	childCriticalErrorReaction : CHILD_CRITICAL_ERROR_REACTION;
	
	i : INT;
		
	child : IChildAutomationComponent;	

	inputDevice : IInputLeafAutomationComponent;
END_VAR
__TRY
	OnBeforeChildrenProcessInput();
__CATCH(exceptionCode)		
	exception := TOF_Core.ExceptionManager.GetLastException(
		exceptionCode := exceptionCode,
		catchPointNamespaceName := NamespaceName,
		catchPointPOUName := __POUNAME(),
		catchPointPosition := __POSITION()
	);
					
	exceptionReaction := OnHandleException(exception := exception, failedMethodName := 'OnBeforeChildrenProcessInput');

	ProcessException(
		exception := exception,
		exceptionReaction := exceptionReaction,
		exceptionSourceHint := "OnBeforeChildrenProcessInput error"
	);
__ENDTRY

FOR i := 0 TO _ChildCount - 1 DO
	child := TryGetChildByIndex(index := i);

	IF child = 0 OR_ELSE NOT child.Enabled OR_ELSE NOT __QUERYINTERFACE(child, inputDevice) THEN
		CONTINUE;
	END_IF
	
	inputDevice.ProcessInput();

	IF inputDevice.HasError AND_THEN inputDevice.Error.Severity = TOF_Core.ERROR_SEVERITY.CRITICAL THEN
		childCriticalErrorReaction := HandleChildCriticalError(childWithError := inputDevice);
		
		ProcessChildError(
			childError := inputDevice.Error,
			childErrorReaction := childCriticalErrorReaction,
			childErrorSourceHint := TOF_Core.WideStrings.Concat255(
				"Child[",
				TO_WSTRING(i),
				"](",
				inputDevice.Name,
				").ProcessInput error"
			)
		);
	END_IF		
END_FOR

__TRY
	OnAfterChildrenProcessInput();
__CATCH(exceptionCode)		
	exception := TOF_Core.ExceptionManager.GetLastException(
		exceptionCode := exceptionCode,
		catchPointNamespaceName := NamespaceName,
		catchPointPOUName := __POUNAME(),
		catchPointPosition := __POSITION()
	);
					
	exceptionReaction := OnHandleException(exception := exception, failedMethodName := 'OnAfterChildrenProcessInput');

	ProcessException(
		exception := exception,
		exceptionReaction := exceptionReaction,
		exceptionSourceHint := "OnAfterChildrenProcessInput error"
	);
__ENDTRY
END_METHOD

(*!
<summary>Processes enabled output children in slot order.</summary>
<description>
A state transition during output processing skips remaining outputs and the after-output hook.
Completed writes remain effective. A pass started in STOPPED proceeds while the branch stays in that state.
</description>
*)
METHOD FINAL ProcessOutput
VAR
	entryRevision : UDINT;
	exceptionCode : __SYSTEM.ExceptionCode;
	exception : TOF_Core.IException;	
	exceptionReaction : TOF_Core.EXCEPTION_REACTION;
	
	childCriticalErrorReaction : CHILD_CRITICAL_ERROR_REACTION;
	
	i : INT;
		
	child : IChildAutomationComponent;	

	outputDevice : IOutputLeafAutomationComponent;
END_VAR
entryRevision := _OperationalStateRevision;

__TRY
	OnBeforeChildrenProcessOutput();
__CATCH(exceptionCode)		
	exception := TOF_Core.ExceptionManager.GetLastException(
		exceptionCode := exceptionCode,
		catchPointNamespaceName := NamespaceName,
		catchPointPOUName := __POUNAME(),
		catchPointPosition := __POSITION()
	);
					
	exceptionReaction := OnHandleException(exception := exception, failedMethodName := 'OnBeforeChildrenProcessOutput');

	ProcessException(
		exception := exception,
		exceptionReaction := exceptionReaction,
		exceptionSourceHint := "OnBeforeChildrenProcessOutput error"
	);
__ENDTRY

FOR i := 0 TO _ChildCount - 1 DO
	IF _OperationalStateRevision <> entryRevision THEN
		RETURN;
	END_IF

	child := TryGetChildByIndex(index := i);

	IF child = 0 OR_ELSE NOT child.Enabled OR_ELSE NOT __QUERYINTERFACE(child, outputDevice) THEN
		CONTINUE;
	END_IF
	
	IF _OperationalStateRevision <> entryRevision THEN
		RETURN;
	END_IF

	outputDevice.ProcessOutput();
	
	IF outputDevice.HasError AND_THEN outputDevice.Error.Severity = TOF_Core.ERROR_SEVERITY.CRITICAL THEN
		childCriticalErrorReaction := HandleChildCriticalError(childWithError := outputDevice);
		
		ProcessChildError(
			childError := outputDevice.Error,
			childErrorReaction := childCriticalErrorReaction,
			childErrorSourceHint := TOF_Core.WideStrings.Concat255(
				"Child[",
				TO_WSTRING(i),
				"](",
				outputDevice.Name,
				").ProcessOutput error"
			)
		);
	END_IF
END_FOR

IF _OperationalStateRevision <> entryRevision THEN
	RETURN;
END_IF

__TRY
	OnAfterChildrenProcessOutput();
__CATCH(exceptionCode)		
	exception := TOF_Core.ExceptionManager.GetLastException(
		exceptionCode := exceptionCode,
		catchPointNamespaceName := NamespaceName,
		catchPointPOUName := __POUNAME(),
		catchPointPosition := __POSITION()
	);
					
	exceptionReaction := OnHandleException(exception := exception, failedMethodName := 'OnAfterChildrenProcessOutput');

	ProcessException(
		exception := exception,
		exceptionReaction := exceptionReaction,
		exceptionSourceHint := "OnAfterChildrenProcessOutput error"
	);
__ENDTRY
END_METHOD

(*!
<summary>Returns a borrowed child by its zero-based index.</summary>
<description>
Returns null when the entry is unavailable, the index is out of range or a nested call raises an exception.
Fatal allocation observations before or after the storage getter return null and preserve the latch for
the outer task boundary. Does not transfer ownership or extend lifetime. Getter exceptions are contained.
</description>
*)
METHOD FINAL TryGetChildByIndex : IChildAutomationComponent
VAR_INPUT
	index : TOF_Core.INT_INDEX;
END_VAR
VAR
	childStorage : REFERENCE TO ARRAY [0.._ChildCount - 1] OF IChildAutomationComponent;
END_VAR
__TRY
	IF TOF_Core.DynamicMemoryManager.HasAllocationFailed OR_ELSE index < 0 OR_ELSE index >= _ChildCount THEN
		RETURN;
	END_IF

	childStorage REF= Children;

	IF NOT TOF_Core.DynamicMemoryManager.HasAllocationFailed AND_THEN __ISVALIDREF(childStorage) THEN
		TryGetChildByIndex := childStorage[index];
	END_IF
__CATCH
	TryGetChildByIndex := 0;
__ENDTRY

IF TOF_Core.DynamicMemoryManager.HasAllocationFailed THEN
	TryGetChildByIndex := 0;
END_IF
END_METHOD

METHOD PROTECTED FINAL Validate
VAR
END_VAR
IF _Parent = 0 THEN
	TOF_Core.Exceptions.ThrowDataMemberNotSpecified(
		sourceNamespaceName := NamespaceName,
		sourceClassName := ClassName,
		sourcePOUName := __POUNAME(),
		sourcePosition := __POSITION(),
		dataMemberName := 'Parent'
	);						
END_IF

IF ChildCount > 0 AND_THEN NOT __ISVALIDREF(Children) THEN
	TOF_Core.Exceptions.ThrowDataMemberNotSpecified(
		sourceNamespaceName := NamespaceName,
		sourceClassName := ClassName,
		sourcePOUName := __POUNAME(),
		sourcePosition := __POSITION(),
		dataMemberName := 'Children'
	);
END_IF
END_METHOD

END_FUNCTION_BLOCK

// ---- AutomationComponent/Branches/ChildCriticalErrorHandlingPolicies/ChildCriticalErrorHandlingPolicies.TcPOU
(*
SPDX-FileCopyrightText: Â© 2026 Oleksandr Tiutyk <trofimich@gmail.com>
SPDX-License-Identifier: MIT
License: https://opensource.org/license/mit
*)

(*!
<summary>Provides shared singleton instances of child critical error handling policies.</summary>
*)

{attribute 'no_explicit_call' := 'do not call this function block directly'}
PROGRAM ChildCriticalErrorHandlingPolicies
VAR
	{attribute 'hide'} 
	_ClassName : STRING := __POUNAME();
	
	{attribute 'hide'} 
	_SetErrorAndStop : SetErrorAndStopAfterCriticalChildErrorHandlingPolicy; 
	{attribute 'hide'} 
	_SetErrorAndContinue : SetErrorAndContinueAfterChildCriticalErrorHandlingPolicy; 
	{attribute 'hide'} 
	_Ignore : IgnoreChildCriticalErrorHandlingPolicy; 
END_VAR

(*!
<summary>Gets the class name of the program.</summary>
*)
{attribute 'monitoring' := 'call'}
PROPERTY ClassName : REFERENCE TO STRING
GET
ClassName REF= _ClassName;
END_GET
END_PROPERTY

(*!
<summary>Gets a shared instance of the ignore error policy.</summary>
*)
{attribute 'monitoring' := 'call'}
PROPERTY Ignore : IChildCriticalErrorHandlingPolicy
GET
Ignore := _Ignore;
END_GET
END_PROPERTY

(*!
<summary>Gets the namespace of the program.</summary>
*)
{attribute 'monitoring' := 'call'}
PROPERTY NamespaceName : REFERENCE TO STRING
GET
NamespaceName REF= CurrentNamespace.Name;
END_GET
END_PROPERTY

(*!
<summary>Gets a shared instance of the set error and continue policy.</summary>
*)
{attribute 'monitoring' := 'call'}
PROPERTY SetErrorAndContinue : IChildCriticalErrorHandlingPolicy
GET
SetErrorAndContinue := _SetErrorAndContinue;
END_GET
END_PROPERTY

(*!
<summary>Gets a shared instance of the set error and stop policy.</summary>
*)
{attribute 'monitoring' := 'call'}
PROPERTY SetErrorAndStop : IChildCriticalErrorHandlingPolicy
GET
SetErrorAndStop := _SetErrorAndStop;
END_GET
END_PROPERTY

END_PROGRAM

// ---- AutomationComponent/Branches/ChildCriticalErrorHandlingPolicies/SetErrorAndStopAfterCriticalChildErrorHandlingPolicy.TcPOU
(*
SPDX-FileCopyrightText: Â© 2026 Oleksandr Tiutyk <trofimich@gmail.com>
SPDX-License-Identifier: MIT
License: https://opensource.org/license/mit
*)

(*!
<summary>Policy that sets parent error and stops execution.</summary>
<description>
Returns CHILD_CRITICAL_ERROR_REACTION.SET_ERROR_AND_STOP when a child component fails.
</description>
*)

{attribute 'no_explicit_call' := 'do not call this function block directly'}
FUNCTION_BLOCK SetErrorAndStopAfterCriticalChildErrorHandlingPolicy EXTENDS TOF_Core.Object IMPLEMENTS IChildCriticalErrorHandlingPolicy
VAR_STAT
	{attribute 'hide'} 
	_ClassName : STRING := __POUNAME();
END_VAR

(*!
<summary>Gets the class name of the policy.</summary>
*)
{attribute 'monitoring' := 'call'}
PROPERTY ClassName : REFERENCE TO STRING
GET
ClassName REF= _ClassName;
END_GET
END_PROPERTY

(*!
<summary>Returns CHILD_CRITICAL_ERROR_REACTION.SET_ERROR_AND_STOP for the child error.</summary>
<param name="childWithError">Child component that reported the error.</param>
<param name="handlingObject">Parent component handling the failure.</param>
*)
METHOD HandleChildCriticalError : CHILD_CRITICAL_ERROR_REACTION
VAR_INPUT
	childWithError : IChildAutomationComponent;
	handlingObject : TOF_Core.IObject;
END_VAR
HandleChildCriticalError := CHILD_CRITICAL_ERROR_REACTION.SET_ERROR_AND_STOP;
END_METHOD

(*!
<summary>Gets the namespace of the policy.</summary>
*)
{attribute 'monitoring' := 'call'}
PROPERTY NamespaceName : REFERENCE TO STRING
GET
NamespaceName REF= CurrentNamespace.Name;
END_GET
END_PROPERTY

(*!
<summary>Gets instance memory footprint in bytes.</summary>
*)
{attribute 'monitoring' := 'call'}
PROPERTY SelfSize : ULINT
GET
SelfSize := XSIZEOF(THIS^);
END_GET
END_PROPERTY

END_FUNCTION_BLOCK

// ---- AutomationComponent/Branches/ChildCriticalErrorHandlingPolicies/SetErrorAndContinueAfterChildCriticalErrorHandlingPolicy.TcPOU
(*
SPDX-FileCopyrightText: Â© 2026 Oleksandr Tiutyk <trofimich@gmail.com>
SPDX-License-Identifier: MIT
License: https://opensource.org/license/mit
*)

(*!
<summary>Policy that sets parent error but continues cyclic execution.</summary>
<description>
Returns CHILD_CRITICAL_ERROR_REACTION.SET_ERROR_AND_CONTINUE when a child component fails.
</description>
*)

{attribute 'no_explicit_call' := 'do not call this function block directly'}
FUNCTION_BLOCK SetErrorAndContinueAfterChildCriticalErrorHandlingPolicy EXTENDS TOF_Core.Object IMPLEMENTS IChildCriticalErrorHandlingPolicy
VAR_STAT
	{attribute 'hide'} 
	_ClassName : STRING := __POUNAME();
END_VAR

(*!
<summary>Gets the class name of the policy.</summary>
*)
{attribute 'monitoring' := 'call'}
PROPERTY ClassName : REFERENCE TO STRING
GET
ClassName REF= _ClassName;
END_GET
END_PROPERTY

(*!
<summary>Returns CHILD_CRITICAL_ERROR_REACTION.SET_ERROR_AND_CONTINUE for the child error.</summary>
<param name="childWithError">Child component that reported the error.</param>
<param name="handlingObject">Parent component handling the failure.</param>
*)
METHOD HandleChildCriticalError : CHILD_CRITICAL_ERROR_REACTION
VAR_INPUT
	childWithError : IChildAutomationComponent;
	handlingObject : TOF_Core.IObject;
END_VAR
HandleChildCriticalError := CHILD_CRITICAL_ERROR_REACTION.SET_ERROR_AND_CONTINUE;
END_METHOD

(*!
<summary>Gets the namespace of the policy.</summary>
*)
{attribute 'monitoring' := 'call'}
PROPERTY NamespaceName : REFERENCE TO STRING
GET
NamespaceName REF= CurrentNamespace.Name;
END_GET
END_PROPERTY

(*!
<summary>Gets instance memory footprint in bytes.</summary>
*)
{attribute 'monitoring' := 'call'}
PROPERTY SelfSize : ULINT
GET
SelfSize := XSIZEOF(THIS^);
END_GET
END_PROPERTY

END_FUNCTION_BLOCK

// ---- AutomationComponent/Branches/ChildCriticalErrorHandlingPolicies/IgnoreChildCriticalErrorHandlingPolicy.TcPOU
(*
SPDX-FileCopyrightText: Â© 2026 Oleksandr Tiutyk <trofimich@gmail.com>
SPDX-License-Identifier: MIT
License: https://opensource.org/license/mit
*)

(*!
<summary>Policy that ignores child critical errors.</summary>
<description>
Returns CHILD_CRITICAL_ERROR_REACTION.IGNORE, allowing the parent component to continue running without error.
</description>
*)

{attribute 'no_explicit_call' := 'do not call this function block directly'}
FUNCTION_BLOCK IgnoreChildCriticalErrorHandlingPolicy EXTENDS TOF_Core.Object IMPLEMENTS IChildCriticalErrorHandlingPolicy
VAR_STAT
	{attribute 'hide'} 
	_ClassName : STRING := __POUNAME();
END_VAR

(*!
<summary>Gets the class name of the policy.</summary>
*)
{attribute 'monitoring' := 'call'}
PROPERTY ClassName : REFERENCE TO STRING
GET
ClassName REF= _ClassName;
END_GET
END_PROPERTY

(*!
<summary>Returns CHILD_CRITICAL_ERROR_REACTION.IGNORE for the child error.</summary>
<param name="childWithError">Child component that reported the error.</param>
<param name="handlingObject">Parent component handling the failure.</param>
*)
METHOD HandleChildCriticalError : CHILD_CRITICAL_ERROR_REACTION
VAR_INPUT
	childWithError : IChildAutomationComponent;
	handlingObject : TOF_Core.IObject;
END_VAR
HandleChildCriticalError := CHILD_CRITICAL_ERROR_REACTION.IGNORE;
END_METHOD

(*!
<summary>Gets the namespace of the policy.</summary>
*)
{attribute 'monitoring' := 'call'}
PROPERTY NamespaceName : REFERENCE TO STRING
GET
NamespaceName REF= CurrentNamespace.Name;
END_GET
END_PROPERTY

(*!
<summary>Gets instance memory footprint in bytes.</summary>
*)
{attribute 'monitoring' := 'call'}
PROPERTY SelfSize : ULINT
GET
SelfSize := XSIZEOF(THIS^);
END_GET
END_PROPERTY

END_FUNCTION_BLOCK

// ---- AutomationComponent/Leafs/InputOutput/InputOutputLeafAutomationComponent.TcPOU
(*
SPDX-FileCopyrightText: Â© 2026 Oleksandr Tiutyk <trofimich@gmail.com>
SPDX-License-Identifier: MIT
License: https://opensource.org/license/mit
*)

(*!
<summary>Base leaf automation component providing both cyclic input and output processing.</summary>
<description>
Derived components override OnProcessInput and OnProcessOutput to interact with field devices.
ProcessInput and ProcessOutput execute the hooks within guarded TRY/CATCH blocks.
</description>
*)

FUNCTION_BLOCK ABSTRACT InputOutputLeafAutomationComponent EXTENDS LeafAutomationComponent
	IMPLEMENTS IInputLeafAutomationComponent, IOutputLeafAutomationComponent

(*!
<summary>Override to perform cyclic reading of input data.</summary>
*)
METHOD PROTECTED ABSTRACT OnProcessInput
END_METHOD

(*!
<summary>Override to perform cyclic writing of output data.</summary>
*)
METHOD PROTECTED ABSTRACT OnProcessOutput
END_METHOD

(*!
<summary>Invokes OnProcessInput with standardized exception handling and error dispatching.</summary>
*)
METHOD FINAL ProcessInput
VAR
	exceptionCode : __SYSTEM.ExceptionCode;
	exception : TOF_Core.IException;
	exceptionReaction : TOF_Core.EXCEPTION_REACTION;
END_VAR
__TRY
	OnProcessInput();
__CATCH(exceptionCode)		
	exception := TOF_Core.ExceptionManager.GetLastException(
		exceptionCode := exceptionCode,
		catchPointNamespaceName := NamespaceName,
		catchPointPOUName := __POUNAME(),
		catchPointPosition := __POSITION()
	);
					
	exceptionReaction := OnHandleException(exception := exception, failedMethodName := 'OnProcessInput');

	ProcessException(
		exception := exception,
		exceptionReaction := exceptionReaction,
		exceptionSourceHint := "OnProcessInput error"
	);
__ENDTRY
END_METHOD

(*!
<summary>Invokes OnProcessOutput with standardized exception handling and error dispatching.</summary>
*)
METHOD FINAL ProcessOutput
VAR
	exceptionCode : __SYSTEM.ExceptionCode;
	exception : TOF_Core.IException;
	exceptionReaction : TOF_Core.EXCEPTION_REACTION;
END_VAR
__TRY
	OnProcessOutput();
__CATCH(exceptionCode)		
	exception := TOF_Core.ExceptionManager.GetLastException(
		exceptionCode := exceptionCode,
		catchPointNamespaceName := NamespaceName,
		catchPointPOUName := __POUNAME(),
		catchPointPosition := __POSITION()
	);
					
	exceptionReaction := OnHandleException(exception := exception, failedMethodName := 'OnProcessOutput');

	ProcessException(
		exception := exception,
		exceptionReaction := exceptionReaction,
		exceptionSourceHint := "OnProcessOutput error"
	);
__ENDTRY
END_METHOD

END_FUNCTION_BLOCK

// ---- AutomationComponent/Leafs/LeafAutomationComponent.TcPOU
(*
SPDX-FileCopyrightText: © 2026 Oleksandr Tiutyk <trofimich@gmail.com>
SPDX-License-Identifier: MIT
License: https://opensource.org/license/mit
*)

(*!
<summary>Base automation component representing a leaf node in the component hierarchy.</summary>
<description>
Leaf components have no children and represent terminal devices, sensors, or actuators.
Events received at this level bubble upwards to the parent component unless propagation is stopped.
Lifecycle methods execute leaf-specific state transitions and invoke overridable hooks. Parent is mandatory
and borrowed for the leaf lifetime. It is checked before initialization hooks. Use one owner task per instance.
Execute() can recover the stored non-critical execution error. Descendants can defer recovery until its
cause clears and can report other diagnostics independently.
</description>
*)

FUNCTION_BLOCK ABSTRACT LeafAutomationComponent EXTENDS AutomationComponent IMPLEMENTS IChildAutomationComponent
VAR
	{attribute 'hide'} 
	_Parent : IParentAutomationComponent;
END_VAR

(*!
<summary>Dispatches event locally and bubbles it up to the parent component.</summary>
<param name="event">The event to dispatch.</param>
*)
METHOD FINAL BubbleEvent
VAR_INPUT
	event : TOF_Core.IEvent;
END_VAR
VAR
	stopPropagation : BOOL;
	
	parentAsBubbleEventDispatcher : TOF_Core.IBubbleEventDispatcher;
END_VAR
OnEventReceived(event := event, stopPropagation => stopPropagation);

IF stopPropagation THEN
	RETURN;
END_IF

IF __QUERYINTERFACE(Parent, parentAsBubbleEventDispatcher) THEN
	parentAsBubbleEventDispatcher.BubbleEvent(event := event);
END_IF
END_METHOD

(*!
<summary>Reports whether Execute() can clear a pending non-critical execution error.</summary>
<description>
The base allows immediate recovery. A descendant can defer recovery by returning FALSE. Execute() calls
this only in WORKING with an active non-critical execution error. Returning FALSE retains the diagnostic
and allows OnWorking to run. Overrides must observe current state without side effects or exceptions.
</description>
*)
METHOD PROTECTED CanRecoverExecutionError : BOOL
CanRecoverExecutionError := TRUE;
END_METHOD

(*!
<summary>Disables the leaf component and invokes OnDisable.</summary>
*)
METHOD FINAL Disable
VAR
	exceptionCode : __SYSTEM.ExceptionCode;
END_VAR
VAR_INST
	disabling : BOOL;
END_VAR
IF NOT _Enabled OR_ELSE disabling THEN
	RETURN;
END_IF

disabling := TRUE;

__TRY
	OnDisable();
	
	_Enabled := FALSE;
	
	disabling := FALSE;	
__CATCH(exceptionCode)
	disabling := FALSE;
	
	TOF_Core.ExceptionManager.ReThrowLastException(
		exceptionCode := exceptionCode,
		catchPointNamespaceName := NamespaceName,
		catchPointPOUName := __POUNAME(),
		catchPointPosition := __POSITION()
	);
__ENDTRY
END_METHOD

(*!
<summary>Enables the leaf component and invokes OnEnable.</summary>
<description>
Enabling does not automatically reset a STOPPED leaf; a disabled stopped leaf remains STOPPED after Enable
until explicitly Reset. If the parent is disabled, enables the parent with includeChildren := FALSE.
</description>
<param name="includeChildren">Ignored for leaf components as they have no children.</param>
*)
METHOD FINAL Enable
VAR_INPUT
	includeChildren : BOOL := TRUE;
END_VAR
VAR
	exceptionCode : __SYSTEM.ExceptionCode;
END_VAR
VAR_INST
	enabling : BOOL;
END_VAR
IF _Enabled OR_ELSE enabling THEN
	RETURN;
END_IF

enabling := TRUE;

__TRY
	OnEnable();
	
	IF _Parent <> 0 AND_THEN NOT _Parent.Enabled THEN
		_Parent.Enable(includeChildren := FALSE);
	END_IF
	
	_Enabled := TRUE;
	
	enabling := FALSE;
__CATCH(exceptionCode)
	enabling := FALSE;
	
	TOF_Core.ExceptionManager.ReThrowLastException(
		exceptionCode := exceptionCode,
		catchPointNamespaceName := NamespaceName,
		catchPointPOUName := __POUNAME(),
		catchPointPosition := __POSITION()
	);
__ENDTRY
END_METHOD

(*!
<summary>Advances cyclic execution for an enabled WORKING or STOPPED leaf.</summary>
<description>
In WORKING, checks CanRecoverExecutionError() for a pending non-critical execution error. When ready,
clears that record and invokes OnRecover before OnWorking. An exception during recovery always records
a copied CRITICAL error, stops the leaf without consulting ExceptionHandlingPolicy, and skips OnWorking.
In STOPPED, invokes OnStopped on each Execute call and logs failures.
</description>
*)
{attribute 'estimated-stack-usage' := '99'}
METHOD FINAL Execute
VAR
	exceptionCode : __SYSTEM.ExceptionCode;
	exception : TOF_Core.IException;	
	exceptionReaction : TOF_Core.EXCEPTION_REACTION;
END_VAR

IF NOT Enabled
	OR_ELSE (_OperationalState <> OPERATIONAL_STATE.WORKING AND_THEN _OperationalState <> OPERATIONAL_STATE.STOPPED)
THEN
	RETURN;
END_IF

CASE _OperationalState OF
	OPERATIONAL_STATE.WORKING:
		IF _Error.HasError AND_THEN _Error.Severity <> TOF_Core.ERROR_SEVERITY.CRITICAL THEN
			__TRY
				IF CanRecoverExecutionError() THEN
					_Error.Clear();
					OnRecover();
				END_IF
			__CATCH(exceptionCode)		
				exception := TOF_Core.ExceptionManager.GetLastException(
					exceptionCode := exceptionCode,
					catchPointNamespaceName := NamespaceName,
					catchPointPOUName := __POUNAME(),
					catchPointPosition := __POSITION()
				);

				// A recovery failure stops the leaf with a critical error without consulting the policy.
				ProcessException(
					exception := exception,
					exceptionReaction := TOF_Core.EXCEPTION_REACTION.SET_ERROR_AND_STOP,
					exceptionSourceHint := "OnRecover error"
				);

				RETURN;
			__ENDTRY
		END_IF
		
		__TRY
			OnWorking();
		__CATCH(exceptionCode)
			exception := TOF_Core.ExceptionManager.GetLastException(
				exceptionCode := exceptionCode,
				catchPointNamespaceName := NamespaceName,
				catchPointPOUName := __POUNAME(),
				catchPointPosition := __POSITION()
			);	
		
			exceptionReaction := OnHandleException(exception := exception, failedMethodName := 'OnWorking');
		
			ProcessException(
				exception := exception,
				exceptionReaction := exceptionReaction,
				exceptionSourceHint := "OnWorking error"
			);
		
			IF exceptionReaction = TOF_Core.EXCEPTION_REACTION.SET_ERROR_AND_STOP THEN
				RETURN;		
			END_IF
		__ENDTRY
		
	OPERATIONAL_STATE.STOPPED:
		__TRY
			OnStopped();
		__CATCH(exceptionCode)
			exception := TOF_Core.ExceptionManager.GetLastException(
				exceptionCode := exceptionCode,
				catchPointNamespaceName := NamespaceName,
				catchPointPOUName := __POUNAME(),
				catchPointPosition := __POSITION()
			);	
		
			exceptionReaction := OnHandleException(exception := exception, failedMethodName := 'OnStopped');
		
			TOF_Core.LogManager.TryLogException(
				exception := exception,
				severity := GetErrorSeverityByExceptionReaction(exceptionReaction := exceptionReaction),
				topic1 := "AutomationComponent",
				topic2 := "AutomationComponent.OnStopped"
			);
		__ENDTRY	
END_CASE
END_METHOD

(*!
<summary>Initializes a new instance of the leaf component.</summary>
<param name="name">Descriptive name of the component.</param>
<param name="parent">Parent automation component in the hierarchy.</param>
*)
METHOD FB_init : BOOL
VAR_INPUT
	bInitRetains : BOOL; // TRUE: the retain variables are initialized (reset warm / reset cold)
	bInCopyCode : BOOL;  // TRUE: the instance will be copied to the copy code afterward (online change)
	name : WSTRING;
	parent : IParentAutomationComponent;
END_VAR
_Parent := parent;
END_METHOD

(*!
<summary>Validates the parent and advances leaf-specific initialization.</summary>
<description>
Parent is mandatory and borrowed for the leaf lifetime. Missing Parent fails before OnInitializing,
even if that hook would complete immediately. FALSE reports pending work or a caught failure; failures
record a critical error in terminal INVALID. TRUE reports completed initialization, including an already
stopped leaf. Completed hook effects are not rolled back.
</description>
*)
METHOD FINAL Initialize : BOOL
VAR
	exceptionCode : __SYSTEM.ExceptionCode;
	exception : TOF_Core.IException;
	
END_VAR
IF _OperationalState <> OPERATIONAL_STATE.INITIALIZING THEN
	Initialize := _OperationalState <> OPERATIONAL_STATE.INVALID;
	
	RETURN;
END_IF

__TRY
	IF _Parent = 0 THEN
		TOF_Core.Exceptions.ThrowDataMemberNotSpecified(
			sourceNamespaceName := NamespaceName,
			sourceClassName := ClassName,
			sourcePOUName := __POUNAME(),
			sourcePosition := __POSITION(),
			dataMemberName := 'Parent'
		);
	END_IF

	Initialize := OnInitializing();
	
	IF Initialize THEN
		SetOperationalState(state := OPERATIONAL_STATE.WORKING, reason := "Successfull initialization");
	ELSE
		IF _InitializationTimer.PT = T#0S THEN
			_InitializationTimer.PT := Parameters.InitializationTimeout;
		END_IF
		
		_InitializationTimer(IN := TRUE);
		
		IF _InitializationTimer.Q THEN		
			TOF_Core.Exceptions.ThrowTimeout(
				sourceNamespaceName := NamespaceName,
				sourceClassName := ClassName,
				sourcePOUName := __POUNAME(),
				sourcePosition := __POSITION(),
				timeoutValue := _InitializationTimer.PT,
				operationName := "Initialization"
			);
		END_IF
		
	END_IF	
__CATCH(exceptionCode)
	Initialize := FALSE;

	exception := TOF_Core.ExceptionManager.GetLastException(
		exceptionCode := exceptionCode,
		catchPointNamespaceName := NamespaceName,
		catchPointPOUName := __POUNAME(),
		catchPointPosition := __POSITION()
	);
	
	ProcessException(
		exception := exception,
		exceptionReaction := TOF_Core.EXCEPTION_REACTION.SET_ERROR_AND_CONTINUE,
		exceptionSourceHint := "Initialization error"
	);					
__ENDTRY
END_METHOD

(*!
<summary>Hook invoked when the leaf component is disabled.</summary>
*)
METHOD PROTECTED OnDisable
END_METHOD

(*!
<summary>Hook invoked when the leaf component is enabled.</summary>
*)
METHOD PROTECTED OnEnable
END_METHOD

(*!
<summary>Hook invoked to perform custom initialization for the leaf component.</summary>
<description>Returns TRUE when initialization completes successfully.</description>
*)
METHOD PROTECTED OnInitializing : BOOL
OnInitializing := TRUE;
END_METHOD

(*!
<summary>Hook invoked when the leaf component is reset from an error state.</summary>
*)
METHOD PROTECTED OnReset
END_METHOD

(*!
<summary>Hook invoked when the leaf component stops execution.</summary>
*)
METHOD PROTECTED OnStopped
END_METHOD

(*!
<summary>Hook invoked during cyclic execution when the leaf component is in the WORKING state.</summary>
*)
METHOD PROTECTED OnWorking
END_METHOD

(*!
<summary>Borrows the constructor-bound parent automation component.</summary>
<description>
Parent is mandatory for initialization and must remain live for the leaf lifetime. The getter does not
transfer ownership or permit reassignment.
</description>
*)
{attribute 'monitoring' := 'call'}
PROPERTY FINAL Parent : IParentAutomationComponent
GET
Parent := _Parent;
END_GET
END_PROPERTY

(*!
<summary>Resets the leaf component from an error state and transitions back to WORKING.</summary>
<description>
Served only while Enabled and STOPPED. Clears the execution error before invoking OnReset. If OnReset raises
an exception, the leaf remains STOPPED with a copied CRITICAL error without consulting ExceptionHandlingPolicy.
Completed hook effects are not rolled back.
</description>
*)
METHOD FINAL Reset
VAR
	exceptionCode : __SYSTEM.ExceptionCode;
	exception : TOF_Core.IException;	
END_VAR
IF NOT Enabled OR_ELSE _OperationalState <> OPERATIONAL_STATE.STOPPED THEN
	RETURN;
END_IF

_Error.Clear();

__TRY
	OnReset();
	
	SetOperationalState(state := OPERATIONAL_STATE.WORKING, reason := "Reset");
__CATCH(exceptionCode)		
	exception := TOF_Core.ExceptionManager.GetLastException(
		exceptionCode := exceptionCode,
		catchPointNamespaceName := NamespaceName,
		catchPointPOUName := __POUNAME(),
		catchPointPosition := __POSITION()
	);

	// A failed reset always keeps the leaf STOPPED with a critical error; the exception policy is not consulted.
	ProcessException(
		exception := exception,
		exceptionReaction := TOF_Core.EXCEPTION_REACTION.SET_ERROR_AND_STOP,
		exceptionSourceHint := "OnReset error"
	);
__ENDTRY
END_METHOD

(*!
<summary>Stops the leaf component and transitions to the STOPPED state.</summary>
<description>
Transitions a WORKING leaf to OPERATIONAL_STATE.STOPPED regardless of Enabled.
</description>
<param name="reason">Descriptive reason for stopping.</param>
*)
METHOD FINAL Stop
VAR_INPUT
	reason : WSTRING(255) := "External stop";
END_VAR
IF _OperationalState <> OPERATIONAL_STATE.WORKING THEN
	RETURN;
END_IF

SetOperationalState(state := OPERATIONAL_STATE.STOPPED, reason := reason);
END_METHOD

END_FUNCTION_BLOCK

// ---- AutomationComponent/Leafs/Input/InputLeafAutomationComponent.TcPOU
(*
SPDX-FileCopyrightText: Â© 2026 Oleksandr Tiutyk <trofimich@gmail.com>
SPDX-License-Identifier: MIT
License: https://opensource.org/license/mit
*)

(*!
<summary>Base leaf automation component providing cyclic input processing.</summary>
<description>
Derived components override OnProcessInput to read inputs from hardware or communications.
ProcessInput executes the hook within a guarded TRY/CATCH block.
</description>
*)

FUNCTION_BLOCK ABSTRACT InputLeafAutomationComponent EXTENDS LeafAutomationComponent
	IMPLEMENTS IInputLeafAutomationComponent

(*!
<summary>Override to perform cyclic reading of input data.</summary>
*)
METHOD PROTECTED ABSTRACT OnProcessInput
END_METHOD

(*!
<summary>Invokes OnProcessInput with standardized exception handling and error dispatching.</summary>
*)
METHOD FINAL ProcessInput
VAR
	exceptionCode : __SYSTEM.ExceptionCode;
	exception : TOF_Core.IException;
	exceptionReaction : TOF_Core.EXCEPTION_REACTION;
END_VAR
__TRY
	OnProcessInput();
__CATCH(exceptionCode)		
	exception := TOF_Core.ExceptionManager.GetLastException(
		exceptionCode := exceptionCode,
		catchPointNamespaceName := NamespaceName,
		catchPointPOUName := __POUNAME(),
		catchPointPosition := __POSITION()
	);
					
	exceptionReaction := OnHandleException(exception := exception, failedMethodName := 'OnProcessInput');

	ProcessException(
		exception := exception,
		exceptionReaction := exceptionReaction,
		exceptionSourceHint := "OnProcessInput error"
	);
__ENDTRY
END_METHOD

END_FUNCTION_BLOCK

// ---- AutomationComponent/Leafs/Output/OutputLeafAutomationComponent.TcPOU
(*
SPDX-FileCopyrightText: Â© 2026 Oleksandr Tiutyk <trofimich@gmail.com>
SPDX-License-Identifier: MIT
License: https://opensource.org/license/mit
*)

(*!
<summary>Base leaf automation component providing cyclic output processing.</summary>
<description>
Derived components override OnProcessOutput to write commands to hardware or actuators.
ProcessOutput executes the hook within a guarded TRY/CATCH block.
</description>
*)

FUNCTION_BLOCK ABSTRACT OutputLeafAutomationComponent EXTENDS LeafAutomationComponent
	IMPLEMENTS IOutputLeafAutomationComponent

(*!
<summary>Override to perform cyclic writing of output data.</summary>
*)
METHOD PROTECTED ABSTRACT OnProcessOutput
END_METHOD

(*!
<summary>Invokes OnProcessOutput with standardized exception handling and error dispatching.</summary>
*)
METHOD FINAL ProcessOutput
VAR
	exceptionCode : __SYSTEM.ExceptionCode;
	exception : TOF_Core.IException;
	exceptionReaction : TOF_Core.EXCEPTION_REACTION;
END_VAR
__TRY
	OnProcessOutput();
__CATCH(exceptionCode)		
	exception := TOF_Core.ExceptionManager.GetLastException(
		exceptionCode := exceptionCode,
		catchPointNamespaceName := NamespaceName,
		catchPointPOUName := __POUNAME(),
		catchPointPosition := __POSITION()
	);
					
	exceptionReaction := OnHandleException(exception := exception, failedMethodName := 'OnProcessOutput');

	ProcessException(
		exception := exception,
		exceptionReaction := exceptionReaction,
		exceptionSourceHint := "OnProcessOutput error"
	);
__ENDTRY
END_METHOD

END_FUNCTION_BLOCK

// ---- AutomationRunner/AutomationRunner.TcPOU
(*
SPDX-FileCopyrightText: © 2026 Oleksandr Tiutyk <trofimich@gmail.com>
SPDX-License-Identifier: MIT
License: https://opensource.org/license/mit
*)

(*!
<summary>Initializes automation components and advances their cyclic execution.</summary>
<description>
FB_init borrows the root array. Its storage and components must outlive all runner calls. Keep its bounds,
slot identities and order fixed. Each root instance must occupy exactly one slot. The runner uses this binding from one task.
Execute updates system services, services the calling task's LogManager destination and processes components
according to the runner state. Its normal epilogue clears the exception payload and releases registered
auto-disposed objects. Call outside handlers that swallow fatal runtime exceptions.
</description>
*)

{attribute 'no_explicit_call' := 'do not call this function block directly'}
FUNCTION_BLOCK AutomationRunner EXTENDS TOF_Core.Object IMPLEMENTS IAutomationRunner
VAR_OUTPUT
	InitializationErrorMessage : TOF_Core.ERROR_MESSAGE;
END_VAR
VAR_STAT
	{attribute 'hide'} 
	_ClassName : STRING := __POUNAME();
END_VAR
VAR
	{attribute 'hide'} 
	_State : AUTOMATION_RUNNER_STATE;
	_Components : POINTER TO IAutomationComponent;
	_FirstIndex : DINT;
	_LastIndex : DINT;
	_RootsValidated : BOOL;
END_VAR

(*!
<summary>Gets the class name of the runner.</summary>
*)
{attribute 'monitoring' := 'call'}
PROPERTY ClassName : REFERENCE TO STRING
GET
ClassName REF= _ClassName;
END_GET
END_PROPERTY

(*!
<summary>Initializes or executes the constructor-bound roots in array order.</summary>
<description>
Once system data is ready, the runner checks the complete root array before initializing any root.
An empty array, null slot or repeated root makes the runner INVALID. Duplicate diagnostics identify both array indices.
Call from the outer task boundary. Nested runner execution is unsupported because cleanup covers the calling task.
Call outside recoverable handlers. Services the current task logger through LogManager.ExecuteCurrentTaskLogger on each call.
A registry allocation failure caught by a callback is raised again at FINAL_ACTIONS.
</description>
*)

METHOD FINAL Execute
VAR
	i : LINT;
	component : IAutomationComponent;
			
	initialized : BOOL;
END_VAR
TOF_Core.System.Execute();		

TOF_Core.LogManager.ExecuteCurrentTaskLogger();

IF TOF_Core.System.SystemDataValid THEN
	CASE _State OF
		AUTOMATION_RUNNER_STATE.INITIALIZING:
			IF NOT _RootsValidated THEN
				InitializationErrorMessage := getRootConfigurationError();

				IF InitializationErrorMessage <> "" THEN
					_State := AUTOMATION_RUNNER_STATE.INVALID;
					JMP FINAL_ACTIONS;
				END_IF

				_RootsValidated := TRUE;
			END_IF

			initialized := TRUE;
			
			FOR i := _FirstIndex TO _LastIndex DO
				component := _Components[TO_UDINT(i - _FirstIndex)];

				IF component = 0 THEN
					_State := AUTOMATION_RUNNER_STATE.INVALID;					
					InitializationErrorMessage := TOF_Core.WideStrings.Concat255("controller[", TO_WSTRING(i), "] is null");					
					JMP FINAL_ACTIONS;					
				END_IF

				component.Initialize();
				
				CASE component.OperationalState OF
					OPERATIONAL_STATE.INVALID:
						_State := AUTOMATION_RUNNER_STATE.INVALID;

						IF TOF_Core.WideStrings.IsNullOrWhiteSpace(stringToCheck := component.OperationalStateReason) THEN
							InitializationErrorMessage := TOF_Core.WideStrings.Concat255(
								"controller[",
								TO_WSTRING(i),
								"] (",
								component.Name,
								") failed"
							);
						ELSE
							InitializationErrorMessage := TOF_Core.WideStrings.Concat255(
								"controller[",
								TO_WSTRING(i),
								"] (",
								component.Name,
								") failed: ",
								component.OperationalStateReason
							);
						END_IF

						JMP FINAL_ACTIONS;
						
					OPERATIONAL_STATE.INITIALIZING:
						initialized := FALSE;						
				END_CASE
			END_FOR		
			
			IF initialized THEN
				_State := AUTOMATION_RUNNER_STATE.RUNNING;
			END_IF
		
		AUTOMATION_RUNNER_STATE.RUNNING:
			FOR i := _FirstIndex TO _LastIndex DO
				component := _Components[TO_UDINT(i - _FirstIndex)];

				IF component <> 0 THEN
					component.Execute();
				END_IF
			END_FOR		
	END_CASE
END_IF

FINAL_ACTIONS:

TOF_Core.DynamicMemoryManager.RaiseIfAllocationFailed();

TOF_Core.ExceptionManager.Cleanup();
TOF_Core.DynamicMemoryManager.CleanupMemory();
END_METHOD

(*!
<summary>Returns the first configuration error in the bound root array, or an empty message on success.</summary>
<description>
Compares interface identities in slot order without invoking root callbacks. Indices use the caller's declared bounds.
</description>
*)
METHOD PRIVATE getRootConfigurationError : WSTRING(255)
VAR
	i : LINT;
	previousIndex : LINT;
	component : IAutomationComponent;
END_VAR
IF _Components = 0 OR_ELSE _LastIndex < _FirstIndex THEN
	getRootConfigurationError := "No controllers to run";
	RETURN;
END_IF

FOR i := _FirstIndex TO _LastIndex DO
	component := _Components[TO_UDINT(i - _FirstIndex)];

	IF component = 0 THEN
		getRootConfigurationError := TOF_Core.WideStrings.Concat255("controller[", TO_WSTRING(i), "] is null");
		RETURN;
	END_IF

	FOR previousIndex := _FirstIndex TO i - 1 DO
		IF _Components[TO_UDINT(previousIndex - _FirstIndex)] = component THEN
			getRootConfigurationError := TOF_Core.WideStrings.Concat255(
				"controller[",
				TO_WSTRING(i),
				"] duplicates controller[",
				TO_WSTRING(previousIndex),
				"]"
			);
			RETURN;
		END_IF
	END_FOR
END_FOR
END_METHOD

(*!
<summary>Binds the runner to the caller's root array for its lifetime.</summary>
<description>
Borrows storage and records the declared index bounds. Root validation and callbacks begin in Execute.
The caller keeps the array and its ordered component references valid for every call.
</description>
<param name="components">Array of automation roots in execution order.</param>
*)
METHOD FB_init : BOOL
VAR_INPUT
	bInitRetains : BOOL; // TRUE: the retain variables are initialized (reset warm / reset cold)
	bInCopyCode : BOOL; // TRUE: the instance will be copied to the copy code afterward (online change)
END_VAR
VAR_IN_OUT CONSTANT
	components : ARRAY [*] OF IAutomationComponent;
END_VAR
_FirstIndex := LOWER_BOUND(components, 1);
_LastIndex := UPPER_BOUND(components, 1);

IF _FirstIndex <= _LastIndex THEN
	_Components := components;
END_IF
END_METHOD

(*!
<summary>Gets the namespace of the runner.</summary>
*)
{attribute 'monitoring' := 'call'}
PROPERTY NamespaceName : REFERENCE TO STRING
GET
NamespaceName REF= CurrentNamespace.Name;
END_GET
END_PROPERTY

(*!
<summary>Gets instance memory footprint in bytes.</summary>
*)
{attribute 'monitoring' := 'call'}
PROPERTY SelfSize : ULINT
GET
SelfSize := XSIZEOF(THIS^);
END_GET
END_PROPERTY

(*!
<summary>Gets current runner state.</summary>
*)
{attribute 'monitoring' := 'call'}
PROPERTY FINAL State : AUTOMATION_RUNNER_STATE
GET
State := _State;
END_GET
END_PROPERTY

(*!
<summary>Gets string representation of current runner state.</summary>
*)
{attribute 'monitoring' := 'call'}
PROPERTY StateName : STRING
GET
StateName := TO_STRING(_State);
END_GET
END_PROPERTY

END_FUNCTION_BLOCK
